FUNCTION_BLOCK RunAxisInspection EXTENDS RunUnitSlave
VAR
	axis1 : POINTER TO RunAxis;
	axis2 : POINTER TO RunAxis;
	sideAligner : POINTER TO RunCylinder := 0;
	
	nCounter : INT := 0;
END_VAR
VAR_OUTPUT
	isLastShot : BOOL;
END_VAR
VAR PERSISTENT
	//Axis1
	indexStandByAxis1 : INT := 1;
	indexPosition1Axis1 : INT := 2;
	//Axis2
	indexStandByAxis2 : INT := 1;
	indexPosition1Axis2 : INT := 2;
	//
	nGoal : INT := 4;
END_VAR

//n-Axis aoi , once position completed , trigger and wait
SUPER^();

CASE outputState OF
	eSpecialStates.SLAVE_AXIS_INSPECTION_ENTER:
		IF NOT transitionByte.0 THEN
			transitionByte.0 := axis1^.ExecuteParameterIndex(nCounter + indexPosition1Axis1);
		END_IF
		IF NOT transitionByte.1 AND_THEN (axis2 = 0 OR (axis2<>0 AND_THEN axis2^.ExecuteParameterIndex(nCounter + indexPosition1Axis2))) THEN
			transitionByte.1 := TRUE; // axis2 is not existed or // axis2 is existed
		END_IF
		IF transitionByte = 3 THEN
			//once inspection done
			NextState := eSpecialStates.SLAVE_AXIS_INSPECTION_ITERATION; //both axis done motion
			slaveWorkingSignal[1] := slaveLinkageStatus[1]; //trigger slave
		END_IF
	eSpecialStates.SLAVE_AXIS_INSPECTION_ITERATION:
		IF NOT slaveWorkingSignal[1] THEN
			//once inspection reach 
			IF nCounter < nGoal THEN			
				nCounter := nCounter + 1;
				NextState := eSpecialStates.SLAVE_AXIS_INSPECTION_ENTER;
			ELSE
				//greater and equal goal
				nCounter := 0; //reset
				NextState := eSpecialStates.SLAVE_AXIS_INSPECTION_EXIT;
			END_IF
		ELSE
			//wait inspecition
		END_IF
END_CASE

//reflect
isLastShot := (nCounter = nGoal);

METHOD FB_init : BOOL
VAR_INPUT
	bInitRetains : BOOL; // if TRUE, the retain variables are initialized (warm start / cold start)
	bInCopyCode : BOOL;  // if TRUE, the instance afterwards gets moved into the copy code (online change)
	
	argParent : POINTER TO RunUnitGeneric;
	argSlotBase : POINTER TO RunMaterial;
	argSlotLast : POINTER TO RunMaterial;
	
	argWorkingSignal : POINTER TO BOOL;
	
	argAxis1 : POINTER TO RunAxis;
	argAxis2 : POINTER TO RunAxis;
	
	argSideAligner : POINTER TO RunCylinder;
END_VAR
//initialize 
Parent := argParent;
SlotBase := argSlotBase;
SlotLast := argSlotLast;
//
IF bInitRetains THEN
	NextState := eSpecialStates.INITIAL_BEGIN;
END_IF

workingSignal := argWorkingSignal; //link

axis1 := argAxis1;
axis2 := argAxis2;
sideAligner := argSideAligner;
END_METHOD

METHOD Initialize : BOOL
VAR_INPUT
END_VAR

//default initialization sequence
CASE outputState OF 
	eSpecialStates.INITIAL_STATE_7:
		IF NOT transitionByte.0 AND_THEN axis1^.ExecuteParameterIndex(indexStandByAxis1) THEN
			transitionByte.0 := TRUE;
		END_IF
		IF NOT transitionByte.1 AND_THEN (axis2 = 0 OR axis2<>0 AND_THEN axis2^.ExecuteParameterIndex(indexStandByAxis2)) THEN
			transitionByte.1 := TRUE; //axis 2 is not existed
		END_IF
		IF NOT transitionByte.2 AND_THEN (sideAligner=0 OR (sideAligner<>0 AND_THEN sideAligner^.Execute(eCylinderCommands.COMMAND_A))) THEN
			transitionByte.2 := TRUE; //aligner backoff
		END_IF
		IF transitionByte = 7 THEN
			NextState := eSpecialStates.INITIAL_END;
		END_IF
END_CASE

Initialize:= SUPER^.Initialize();
END_METHOD

END_FUNCTION_BLOCK

(* stored: Version 1.1.0.1, ProductVersion 3.1.4022.10
   POU RunAxisInspection: Id {a6e0aedf-0dab-4fac-b5f4-4cfe5e671281}, SpecialFunc None
   Method FB_init: Id {d0f76d0d-18fe-401c-ac9e-95df7adf4d63}
   Method Initialize: Id {130164f8-aa24-4f6f-8c9b-a99078376a66} *)
